// TwinCAT 3 PLC project FactoryIO
// ProgramVersion: 3.1.4024.0
// libraries:
//   Tc2_ModbusSrv, * (Beckhoff Automation GmbH)
//   Tc2_Standard, * (Beckhoff Automation GmbH)
//   Tc2_System, * (Beckhoff Automation GmbH)
//   Tc3_Module, * (Beckhoff Automation GmbH)
// project tree:
//   GVLs/ GVL.TcGVL
//   / PlcTask.TcTTO
//   POUs/FBs/Conveyor/DUTs/ E_ConveyorStates.TcDUT, ST_ConveyorConfiguration.TcDUT, ST_ConveyorControls.TcDUT, ST_ConveyorStatus.TcDUT
//   POUs/FBs/Conveyor/ FB_Conveyor.TcPOU
//   POUs/FBs/IndexedPosition/DUTs/ E_IndexedPositionSimplifiedRequest.TcDUT, E_IndexedPositionStates.TcDUT, E_IndexedPositionTransitionRequest.TcDUT, ST_DirectionalControls.TcDUT, ST_IndexedPositionControls.TcDUT, ST_IndexedPositionLinks.TcDUT
//   POUs/FBs/IndexedPosition/ FB_IndexedPosition.TcPOU
//   POUs/FBs/LTU/DUTs/ E_LTUHardwareState.TcDUT, ST_LTUConfiguration.TcDUT, ST_LTUStatus.TcDUT
//   POUs/FBs/LTU/ FB_LTU.TcPOU
//   POUs/FBs/PalletStop/DUTs/ E_PalletStopHardwareStates.TcDUT, ST_PalletStopConfiguration.TcDUT, ST_PalletStopStatus.TcDUT
//   POUs/FBs/PalletStop/ FB_PalletStop.TcPOU
//   POUs/FBs/PartPresence/DUTs/ E_ActivationType.TcDUT, ST_PartPresenceConfiguration.TcDUT, ST_PartPresenceStatus.TcDUT
//   POUs/FBs/PartPresence/ FB_PartPresence.TcPOU
//   POUs/ MAIN.TcPOU
// real-time tasks:
//   TASK PlcTask: cycle T#10ms, priority 20, ADS port 350

CONFIGURATION FactoryIO
    RESOURCE PLC ON TwinCAT3
        TASK PlcTask(INTERVAL := T#10ms, PRIORITY := 20);
        PROGRAM MAIN WITH PlcTask : MAIN;
    END_RESOURCE
END_CONFIGURATION

// ---- POUs/FBs/Conveyor/DUTs/E_ConveyorStates.TcDUT
{attribute 'qualified_only'}
{attribute 'strict'}
TYPE E_ConveyorStates :
(
	Stopped,
	RunRequest,
	Running,
	StopRequest,
	Fault
);
END_TYPE

// ---- POUs/FBs/Conveyor/DUTs/ST_ConveyorConfiguration.TcDUT
TYPE ST_ConveyorConfiguration :
	STRUCT
		Name 				: STRING := 'Conveyor'; 	// Name of the conveyor
		HardwareOutput 		: DINT;						// What position in the TCP/IP array this Bit is connected to for the simulationm
		OutputArrayPosition	: DINT;						// Equal to HardwareOutput - 32768
	END_STRUCT
END_TYPE

// ---- POUs/FBs/Conveyor/DUTs/ST_ConveyorControls.TcDUT
TYPE ST_ConveyorControls :
	STRUCT
		RequestRun 		: BOOL := FALSE; // Requests the conveyance to run
		RequestStop		: BOOL := FALSE; // Requests the conveyance to stop
		OperationMode	: BOOL := FALSE; // TRUE = Automatic, FALSE = Manual 
	END_STRUCT
END_TYPE

// ---- POUs/FBs/Conveyor/DUTs/ST_ConveyorStatus.TcDUT
TYPE ST_ConveyorStatus :
	STRUCT
		isRunning	: BOOL;  // This varriable will be True when the conveyor is running and False when it is not running
	END_STRUCT
END_TYPE

// ---- POUs/FBs/IndexedPosition/DUTs/E_IndexedPositionSimplifiedRequest.TcDUT
{attribute 'qualified_only'}
{attribute 'strict'}
TYPE E_IndexedPositionSimplifiedRequest :
(
	NoRequest,
	Busy,
	Send,
	Recieve
);
END_TYPE

// ---- POUs/FBs/IndexedPosition/DUTs/E_IndexedPositionStates.TcDUT
{attribute 'qualified_only'}
{attribute 'strict'}
TYPE E_IndexedPositionStates :
(
	Starved,
	Idle,
	Blocked,
	ReceivingFromLeft,
	ReceivingFromRight,
	ReceivingFromFront,
	ReceivingFromRear,
	SendingToLeft,
	SendingToRight,
	SendingToFront,
	SendingToRear,
	Bypass,
	Fault
);
END_TYPE

// ---- POUs/FBs/IndexedPosition/DUTs/E_IndexedPositionTransitionRequest.TcDUT
{attribute 'qualified_only'}
{attribute 'strict'}
TYPE E_IndexedPositionTransitionRequest :
(
	NoRequest,
	ReceiveFromLeft,
	ReceiveFromRight,
	ReceiveFromFront,
	ReceiveFromRear,
	SendToLeft,
	SendToRight,
	SendToFront,
	SendToRear
);
END_TYPE

// ---- POUs/FBs/IndexedPosition/DUTs/ST_DirectionalControls.TcDUT
TYPE ST_DirectionalControls :
	STRUCT
		Request 			: E_IndexedPositionSimplifiedRequest;
		PartPresent 		: BOOL;
		State				: E_IndexedPositionStates := E_IndexedPositionStates.Starved;
		OperationMode		: BOOL;
		isDefined 			: BOOL;
	END_STRUCT
END_TYPE

// ---- POUs/FBs/IndexedPosition/DUTs/ST_IndexedPositionControls.TcDUT
TYPE ST_IndexedPositionControls :
	STRUCT
		// Operating modes
		OperationMode		: BOOL := FALSE; // TRUE = Automatic, FALSE = Manual
		isDefined 			: BOOL := FALSE; // Change to true if this position exists
		State				: E_IndexedPositionStates := E_IndexedPositionStates.Starved;
		Request				: E_IndexedPositionTransitionRequest := E_IndexedPositionTransitionRequest.NoRequest;
		
		// Sensing
		ArrivalDetection	: BOOL;
		AreaMonitoring		: BOOL;

		// Internal Directional Controls for Linking
		Front				: ST_DirectionalControls;
		Rear				: ST_DirectionalControls;
		Left				: ST_DirectionalControls;
		Right				: ST_DirectionalControls;
		
	END_STRUCT
END_TYPE

// ---- POUs/FBs/IndexedPosition/DUTs/ST_IndexedPositionLinks.TcDUT
TYPE ST_IndexedPositionLinks :
	STRUCT
		Front				: REFERENCE TO ST_DirectionalControls;
		Rear				: REFERENCE TO ST_DirectionalControls;
		Left				: REFERENCE TO ST_DirectionalControls;
		Right				: REFERENCE TO ST_DirectionalControls;
	END_STRUCT
END_TYPE

// ---- POUs/FBs/LTU/DUTs/E_LTUHardwareState.TcDUT
{attribute 'qualified_only'}
{attribute 'strict'}
TYPE E_LTUHardwareState :
(
	NoCommand,
	RunForward,
	RunReverse,
	RunLeft,
	RunRight
);
END_TYPE

// ---- POUs/FBs/LTU/DUTs/ST_LTUConfiguration.TcDUT
TYPE ST_LTUConfiguration :
	STRUCT
		Name 						: STRING := 'LTU'; 			// Name of the LTU
		
		ForwardHardwareOutput 		: DINT;						// What position in the TCP/IP array this Bit is connected to for the simulationm
		ReverseHardwareOutput 		: DINT;						// What position in the TCP/IP array this Bit is connected to for the simulationm
		LeftHardwareOutput 			: DINT;						// What position in the TCP/IP array this Bit is connected to for the simulationm
		RightHardwareOutput 		: DINT;						// What position in the TCP/IP array this Bit is connected to for the simulationm
		
		ForwardOutputArrayPosition	: DINT;						// Equal to associated HardwareOutput - 32768
		ReverseOutputArrayPosition	: DINT;						// Equal to associated HardwareOutput - 32768
		LeftOutputArrayPosition		: DINT;						// Equal to associated HardwareOutput - 32768
		RightOutputArrayPosition	: DINT;						// Equal to associated HardwareOutput - 32768
		
		BypassLTU					: BOOL := FALSE; 			// This will have the LTU spin forward continuousle
	END_STRUCT
END_TYPE

// ---- POUs/FBs/LTU/DUTs/ST_LTUStatus.TcDUT
TYPE ST_LTUStatus :
STRUCT
END_STRUCT
END_TYPE

// ---- POUs/FBs/PalletStop/DUTs/E_PalletStopHardwareStates.TcDUT
{attribute 'qualified_only'}
{attribute 'strict'}
TYPE E_PalletStopHardwareStates :
(
	Raised,
	Lowered,
	Raising,
	Lowering,
	Fault
);
END_TYPE

// ---- POUs/FBs/PalletStop/DUTs/ST_PalletStopConfiguration.TcDUT
TYPE ST_PalletStopConfiguration :
	STRUCT
		Name 							: STRING := 'PalletStop'; 	// Name of the PalletStop
		DownStreamHardwareOutput 		: DINT;						// What position in the TCP/IP array this Bit is connected to for the simulationm
		DownStreamOutputArrayPosition	: DINT;						// Equal to associated HardwareOutput - 32768
	END_STRUCT
END_TYPE

// ---- POUs/FBs/PalletStop/DUTs/ST_PalletStopStatus.TcDUT
TYPE ST_PalletStopStatus :
	STRUCT
	END_STRUCT
END_TYPE

// ---- POUs/FBs/PartPresence/DUTs/E_ActivationType.TcDUT
{attribute 'qualified_only'}
{attribute 'strict'}
TYPE E_ActivationType :
(
	NormallyOpen,
	NormallyClosed
);
END_TYPE

// ---- POUs/FBs/PartPresence/DUTs/ST_PartPresenceConfiguration.TcDUT
TYPE ST_PartPresenceConfiguration :
	STRUCT
		Name 			: STRING := 'Part Presence';
		ActivationType 	: E_ActivationType := E_ActivationType.NormallyOpen;
		DebounceOnTime	: TIME := T#0S;
		DebounceOffTime	: TIME := T#0S;
		
		HardwareInput 		: BOOL;			// Mapped directly from the array
	END_STRUCT
END_TYPE

// ---- POUs/FBs/PartPresence/DUTs/ST_PartPresenceStatus.TcDUT
TYPE ST_PartPresenceStatus :
	STRUCT
		isOn : BOOL;
	END_STRUCT
END_TYPE

// ---- GVLs/GVL.TcGVL
{attribute 'qualified_only'}
VAR_GLOBAL
	mb_Input_Coils : ARRAY [0..255] OF BOOL;
	mb_Output_Coils : ARRAY [0..255] OF BOOL;
	
	// initializeControls : ST_IndexedPositionControls;
END_VAR

// ---- POUs/MAIN.TcPOU
PROGRAM MAIN
VAR
	// Actuators
	Conveyors		: ARRAY [0..16] OF FB_Conveyor;
	LTUs			: ARRAY [1..6] OF FB_LTU;
	PalletStops		: ARRAY [0..32] OF FB_PalletStop;
	
	// Sensors
	PalletStop_PartPresence_DetectArrival 	: ARRAY [0..32] OF FB_PartPresence;
	PalletStop_PartPresence_AreaMonitor		: ARRAY [0..32] OF FB_PartPresence;
	LTU_PartPresence_DetectArrival 			: ARRAY [1..6] OF FB_PartPresence;
	LTU_PartPresence_AreaMonitor			: ARRAY [1..6] OF FB_PartPresence;
	
	FirstScan		: BOOL := TRUE;
	i				: DINT;
	ToggleOn		: BOOL := FALSE;
	ToggleOff		: BOOL := FALSE;
	arrayOffset		: DINT := 32768;
	
	A : BOOL := FALSE;
END_VAR

// Fill in Reset Methods
// Set up main method for Material Flow
// Set up Error Handling
// Setup Manual Controls
// Create TwinCAT HMI for Manual Controls
// Download free ignition and create scada page
// Add Logic for sensor decisions
// Add an Actuator to do something?
// Save in GIT repo
// Maybe Add Safety and Stack Lights, Safety as real virtual safety
// Difference between HMI anbd SCADA
// Maybe Add Some Ladder?
// Scada part request

M_PartPresenceSensors();
M_Conveyors();
M_PalletStops();
M_LTUs();
M_ConveyanceLogic();

// Conveyors
FOR i := 0 TO 16 BY 1 DO
	IF ToggleOn THEN
		Conveyors[i].P_Controls.RequestRun := TRUE;
	ELSIF ToggleOff THEN
		Conveyors[i].P_Controls.RequestStop := TRUE;
	END_IF
END_FOR
ToggleOn := FALSE;
ToggleOff := FALSE;

FirstScan := FALSE;

METHOD PUBLIC M_ConveyanceLogic : BOOL
VAR_INPUT
END_VAR
///////////////////////////////////////////////////////////////////////////////////////////////////////////////////////////////////
/////////////////////////////////////////////////////// Pallet Stop Linking ///////////////////////////////////////////////////////
///////////////////////////////////////////////////////////////////////////////////////////////////////////////////////////////////

// Pallet Stop 00
PalletStops[0].P_Links.Rear 	REF= PalletStops[31].P_Controls.Front;
PalletStops[0].P_Links.Front	REF= PalletStops[1].P_Controls.Rear;

// Pallet Stop 01
PalletStops[1].P_Links.Rear		REF= PalletStops[0].P_Controls.Front;
PalletStops[1].P_Links.Front 	REF= LTUs[1].P_Controls.Rear;

// Pallet Stop 02
// Skipped

// Pallet Stop 03
PalletStops[3].P_Links.Rear		REF= LTUs[1].P_Controls.Left;
PalletStops[3].P_Links.Front 	REF= PalletStops[4].P_Controls.Rear;

// Pallet Stop 04
PalletStops[4].P_Links.Rear		REF= PalletStops[3].P_Controls.Front;
PalletStops[4].P_Links.Front 	REF= PalletStops[5].P_Controls.Rear;

// Pallet Stop 05
PalletStops[5].P_Links.Rear		REF= PalletStops[4].P_Controls.Front;
PalletStops[5].P_Links.Front 	REF= PalletStops[7].P_Controls.Rear;

// Pallet Stop 06
PalletStops[6].P_Links.Rear		REF= LTUs[1].P_Controls.Front;
PalletStops[6].P_Links.Front 	REF= LTUs[2].P_Controls.Right;

// Pallet Stop 07
PalletStops[7].P_Links.Rear		REF= PalletStops[5].P_Controls.Front;
PalletStops[7].P_Links.Front 	REF= LTUs[2].P_Controls.Rear;

// Pallet Stop 08
// Skipped

// Pallet Stop 09
// Skipped

// Pallet Stop 10
PalletStops[10].P_Links.Rear	REF= LTUs[2].P_Controls.Left;
PalletStops[10].P_Links.Front 	REF= LTUs[3].P_Controls.Rear;;

// Pallet Stop 11
// Skipped

// Pallet Stop 12
PalletStops[12].P_Links.Rear	REF= LTUs[3].P_Controls.Left;
PalletStops[12].P_Links.Front 	REF= LTUs[4].P_Controls.Rear;;

// Pallet Stop 13
// Skipped

// Pallet Stop 14
PalletStops[14].P_Links.Rear	REF= LTUs[4].P_Controls.Right;
PalletStops[14].P_Links.Front 	REF= PalletStops[15].P_Controls.Rear;

// Pallet Stop 15
PalletStops[15].P_Links.Rear	REF= PalletStops[14].P_Controls.Front;
PalletStops[15].P_Links.Front 	REF= PalletStops[16].P_Controls.Rear;

// Pallet Stop 16
PalletStops[16].P_Links.Rear	REF= PalletStops[15].P_Controls.Front;
PalletStops[16].P_Links.Front 	REF= PalletStops[17].P_Controls.Rear;

// Pallet Stop 17
PalletStops[17].P_Links.Rear	REF= PalletStops[16].P_Controls.Front;
PalletStops[17].P_Links.Front 	REF= PalletStops[32].P_Controls.Rear; // 18b

// Pallet Stop 18
PalletStops[18].P_Links.Rear	REF= LTUs[3].P_Controls.Front;
PalletStops[18].P_Links.Front 	REF= LTUs[5].P_Controls.Rear;

// Pallet Stop 19
PalletStops[19].P_Links.Rear	REF= PalletStops[32].P_Controls.Front; // 18b
PalletStops[19].P_Links.Front 	REF= LTUs[6].P_Controls.Left;

// Pallet Stop 20
// Skipped

// Pallet Stop 21
PalletStops[21].P_Links.Rear	REF= LTUs[6].P_Controls.Right;
PalletStops[21].P_Links.Front 	REF= PalletStops[22].P_Controls.Rear;

IF PalletStops[21].P_Controls.ArrivalDetection THEN
	PalletStops[21].P_Controls.Request := E_IndexedPositionTransitionRequest.SendToFront;
	//PalletStops[21].P_Links.Front.Request := E_IndexedPositionTransitionRequest.ReceiveForward;
END_IF

// Pallet Stop 22
PalletStops[22].P_Links.Rear	REF= PalletStops[21].P_Controls.Front;
PalletStops[22].P_Links.Front 	REF= PalletStops[23].P_Controls.Rear;

IF PalletStops[22].P_Controls.ArrivalDetection THEN
	PalletStops[22].P_Controls.Request := E_IndexedPositionTransitionRequest.SendToFront;
	//PalletStops[22].P_Links.Front.Request := E_IndexedPositionTransitionRequest.ReceiveForward;
END_IF

// Pallet Stop 23
PalletStops[23].P_Links.Rear	REF= PalletStops[22].P_Controls.Front;
PalletStops[23].P_Links.Front 	REF= PalletStops[24].P_Controls.Rear;

IF PalletStops[23].P_Controls.ArrivalDetection THEN
	PalletStops[23].P_Controls.Request := E_IndexedPositionTransitionRequest.SendToFront;
	//PalletStops[23].P_Links.Front.Request := E_IndexedPositionTransitionRequest.ReceiveForward;
END_IF

// Pallet Stop 24
PalletStops[24].P_Links.Rear	REF= PalletStops[23].P_Controls.Front;
PalletStops[24].P_Links.Front 	REF= PalletStops[25].P_Controls.Rear;

IF PalletStops[24].P_Controls.ArrivalDetection THEN
	PalletStops[24].P_Controls.Request := E_IndexedPositionTransitionRequest.SendToFront;
	//PalletStops[24].P_Links.Front.Request := E_IndexedPositionTransitionRequest.ReceiveForward;
END_IF

// Pallet Stop 25
PalletStops[25].P_Links.Rear	REF= PalletStops[24].P_Controls.Front;
PalletStops[25].P_Links.Front 	REF= PalletStops[26].P_Controls.Rear;

IF PalletStops[25].P_Controls.ArrivalDetection THEN
	PalletStops[25].P_Controls.Request := E_IndexedPositionTransitionRequest.SendToFront;
	//PalletStops[25].P_Links.Front.Request := E_IndexedPositionTransitionRequest.ReceiveForward;
END_IF

// Pallet Stop 26
PalletStops[26].P_Links.Rear	REF= PalletStops[25].P_Controls.Front;
PalletStops[26].P_Links.Front 	REF= PalletStops[27].P_Controls.Rear;

IF PalletStops[26].P_Controls.ArrivalDetection THEN
	PalletStops[26].P_Controls.Request := E_IndexedPositionTransitionRequest.SendToFront;
	//PalletStops[26].P_Links.Front.Request := E_IndexedPositionTransitionRequest.ReceiveForward;
END_IF

// Pallet Stop 27
PalletStops[27].P_Links.Rear	REF= PalletStops[26].P_Controls.Front;
PalletStops[27].P_Links.Front 	REF= PalletStops[28].P_Controls.Rear;

IF PalletStops[27].P_Controls.ArrivalDetection THEN
	PalletStops[27].P_Controls.Request := E_IndexedPositionTransitionRequest.SendToFront;
	//PalletStops[27].P_Links.Front.Request := E_IndexedPositionTransitionRequest.ReceiveForward;
END_IF

// Pallet Stop 28
PalletStops[28].P_Links.Rear	REF= PalletStops[27].P_Controls.Front;
PalletStops[28].P_Links.Front 	REF= PalletStops[29].P_Controls.Rear;

IF PalletStops[28].P_Controls.ArrivalDetection THEN
	PalletStops[28].P_Controls.Request := E_IndexedPositionTransitionRequest.SendToFront;
	//PalletStops[28].P_Links.Front.Request := E_IndexedPositionTransitionRequest.ReceiveForward;
END_IF

// Pallet Stop 29
PalletStops[29].P_Links.Rear	REF= PalletStops[28].P_Controls.Front;
PalletStops[29].P_Links.Front 	REF= PalletStops[30].P_Controls.Rear;

IF PalletStops[29].P_Controls.ArrivalDetection THEN
	PalletStops[29].P_Controls.Request := E_IndexedPositionTransitionRequest.SendToFront;
	//PalletStops[29].P_Links.Front.Request := E_IndexedPositionTransitionRequest.ReceiveForward;
END_IF

// Pallet Stop 30
PalletStops[30].P_Links.Rear	REF= PalletStops[29].P_Controls.Front;
PalletStops[30].P_Links.Front 	REF= PalletStops[31].P_Controls.Rear;

IF PalletStops[30].P_Controls.ArrivalDetection THEN
	PalletStops[30].P_Controls.Request := E_IndexedPositionTransitionRequest.SendToFront;
	//PalletStops[30].P_Links.Front.Request := E_IndexedPositionTransitionRequest.ReceiveForward;
END_IF

// Pallet Stop 31
PalletStops[31].P_Links.Rear	REF= PalletStops[30].P_Controls.Front;
PalletStops[31].P_Links.Front 	REF= PalletStops[0].P_Controls.Rear;

IF PalletStops[31].P_Controls.ArrivalDetection THEN
	PalletStops[31].P_Controls.Request := E_IndexedPositionTransitionRequest.SendToFront;
	//PalletStops[31].P_Links.Front.Request := E_IndexedPositionTransitionRequest.ReceiveForward;
END_IF

// Pallet Stop 18b
PalletStops[32].P_Links.Rear	REF= PalletStops[17].P_Controls.Front;
PalletStops[32].P_Links.Front 	REF= PalletStops[19].P_Controls.Rear;
END_METHOD

METHOD PUBLIC M_Conveyors : BOOL
VAR_INPUT
END_VAR
IF FirstScan THEN
	// Initialize
	FOR i := 0 TO 16 BY 1 DO
		Conveyors[i].P_Configuration.Name := CONCAT('Conveyor ', DINT_TO_STRING(i));
		Conveyors[i].P_Configuration.HardwareOutput := 32771 + i;
	END_FOR
ELSE
	FOR i := 0 TO 16 BY 1 DO
		Conveyors[i](HardwareInputArray := GVL.mb_Input_Coils);
	END_FOR
END_IF
END_METHOD

METHOD PUBLIC M_LTUs : BOOL
VAR_INPUT
END_VAR
IF FirstScan THEN
	// Initialize
	FOR i := 1 TO 6 BY 1 DO
		LTUs[i].P_Configuration.Name := CONCAT('LTU ', DINT_TO_STRING(i));
		LTUs[i].P_Configuration.ForwardHardwareOutput 	:= 32790 + 1 + ((i-1)*4);
		LTUs[i].P_Configuration.ReverseHardwareOutput 	:= 32790 + 2 + ((i-1)*4);
		LTUs[i].P_Configuration.LeftHardwareOutput 		:= 32790 + 3 + ((i-1)*4);
		LTUs[i].P_Configuration.RightHardwareOutput 	:= 32790 + 4 + ((i-1)*4);
	END_FOR
ELSE
	// Update Area Monitoring and Arrival Detection
	FOR i := 1 TO 6 BY 1 DO
		LTUs[i].P_Controls.AreaMonitoring 		:= LTU_PartPresence_AreaMonitor[i].P_Status.isOn;
		LTUs[i].P_Controls.ArrivalDetection 	:= LTU_PartPresence_DetectArrival[i].P_Status.isOn;
		LTUs[i](HardwareInputArray := GVL.mb_Input_Coils);
	END_FOR
END_IF
END_METHOD

METHOD M_PalletStops : BOOL
VAR_INPUT
END_VAR
IF FirstScan THEN
	// Initialize
	FOR i := 0 TO 32 BY 1 DO
		PalletStops[i].P_Configuration.Name := CONCAT('Pallet Stop ', DINT_TO_STRING(i));
		PalletStops[i].P_Configuration.DownStreamHardwareOutput := 32818 + i;
	END_FOR
ELSE
	// Update Area Monitoring and Arrival Detection
	FOR i := 0 TO 32 BY 1 DO
		PalletStops[i].P_Controls.AreaMonitoring 	:= PalletStop_PartPresence_AreaMonitor[i].P_Status.isOn;
		PalletStops[i].P_Controls.ArrivalDetection 	:= PalletStop_PartPresence_DetectArrival[i].P_Status.isOn;
		PalletStops[i](HardwareInputArray := GVL.mb_Input_Coils);
	END_FOR
END_IF
END_METHOD

METHOD PUBLIC M_PartPresenceSensors : BOOL
PalletStop_PartPresence_DetectArrival[0].P_Configuration.HardwareInput := GVL.mb_Output_Coils[32771 - arrayOffset];
PalletStop_PartPresence_DetectArrival[1].P_Configuration.HardwareInput := GVL.mb_Output_Coils[32772 - arrayOffset];
PalletStop_PartPresence_DetectArrival[2].P_Configuration.HardwareInput := GVL.mb_Output_Coils[32773 - arrayOffset];
PalletStop_PartPresence_DetectArrival[3].P_Configuration.HardwareInput := GVL.mb_Output_Coils[32774 - arrayOffset];
PalletStop_PartPresence_DetectArrival[4].P_Configuration.HardwareInput := GVL.mb_Output_Coils[32775 - arrayOffset];
PalletStop_PartPresence_DetectArrival[5].P_Configuration.HardwareInput := GVL.mb_Output_Coils[32776 - arrayOffset];
PalletStop_PartPresence_DetectArrival[6].P_Configuration.HardwareInput := GVL.mb_Output_Coils[32777 - arrayOffset];
PalletStop_PartPresence_DetectArrival[7].P_Configuration.HardwareInput := GVL.mb_Output_Coils[32778 - arrayOffset];
PalletStop_PartPresence_DetectArrival[8].P_Configuration.HardwareInput := GVL.mb_Output_Coils[32779 - arrayOffset];
PalletStop_PartPresence_DetectArrival[9].P_Configuration.HardwareInput := GVL.mb_Output_Coils[32780 - arrayOffset];
PalletStop_PartPresence_DetectArrival[10].P_Configuration.HardwareInput := GVL.mb_Output_Coils[32781 - arrayOffset];
PalletStop_PartPresence_DetectArrival[11].P_Configuration.HardwareInput := GVL.mb_Output_Coils[32782 - arrayOffset];
PalletStop_PartPresence_DetectArrival[12].P_Configuration.HardwareInput := GVL.mb_Output_Coils[32783 - arrayOffset];
PalletStop_PartPresence_DetectArrival[13].P_Configuration.HardwareInput := GVL.mb_Output_Coils[32784 - arrayOffset];
PalletStop_PartPresence_DetectArrival[14].P_Configuration.HardwareInput := GVL.mb_Output_Coils[32785 - arrayOffset];
PalletStop_PartPresence_DetectArrival[15].P_Configuration.HardwareInput := GVL.mb_Output_Coils[32786 - arrayOffset];
PalletStop_PartPresence_DetectArrival[16].P_Configuration.HardwareInput := GVL.mb_Output_Coils[32787 - arrayOffset];
PalletStop_PartPresence_DetectArrival[17].P_Configuration.HardwareInput := GVL.mb_Output_Coils[32788 - arrayOffset];
PalletStop_PartPresence_DetectArrival[18].P_Configuration.HardwareInput := GVL.mb_Output_Coils[32789 - arrayOffset];
PalletStop_PartPresence_DetectArrival[19].P_Configuration.HardwareInput := GVL.mb_Output_Coils[32790 - arrayOffset];
PalletStop_PartPresence_DetectArrival[20].P_Configuration.HardwareInput := GVL.mb_Output_Coils[32791 - arrayOffset];
PalletStop_PartPresence_DetectArrival[21].P_Configuration.HardwareInput := GVL.mb_Output_Coils[32792 - arrayOffset];
PalletStop_PartPresence_DetectArrival[22].P_Configuration.HardwareInput := GVL.mb_Output_Coils[32793 - arrayOffset];
PalletStop_PartPresence_DetectArrival[23].P_Configuration.HardwareInput := GVL.mb_Output_Coils[32794 - arrayOffset];
PalletStop_PartPresence_DetectArrival[24].P_Configuration.HardwareInput := GVL.mb_Output_Coils[32795 - arrayOffset];
PalletStop_PartPresence_DetectArrival[25].P_Configuration.HardwareInput := GVL.mb_Output_Coils[32796 - arrayOffset];
PalletStop_PartPresence_DetectArrival[26].P_Configuration.HardwareInput := GVL.mb_Output_Coils[32797 - arrayOffset];
PalletStop_PartPresence_DetectArrival[27].P_Configuration.HardwareInput := GVL.mb_Output_Coils[32798 - arrayOffset];
PalletStop_PartPresence_DetectArrival[28].P_Configuration.HardwareInput := GVL.mb_Output_Coils[32799 - arrayOffset];
PalletStop_PartPresence_DetectArrival[29].P_Configuration.HardwareInput := GVL.mb_Output_Coils[32800 - arrayOffset];
PalletStop_PartPresence_DetectArrival[30].P_Configuration.HardwareInput := GVL.mb_Output_Coils[32801 - arrayOffset];
PalletStop_PartPresence_DetectArrival[31].P_Configuration.HardwareInput := GVL.mb_Output_Coils[32802 - arrayOffset];
PalletStop_PartPresence_DetectArrival[32].P_Configuration.HardwareInput := GVL.mb_Output_Coils[32803 - arrayOffset];

PalletStop_PartPresence_AreaMonitor[0].P_Configuration.HardwareInput := GVL.mb_Output_Coils[32807 - arrayOffset];
PalletStop_PartPresence_AreaMonitor[1].P_Configuration.HardwareInput := GVL.mb_Output_Coils[32808 - arrayOffset];
PalletStop_PartPresence_AreaMonitor[2].P_Configuration.HardwareInput := GVL.mb_Output_Coils[32809 - arrayOffset];
PalletStop_PartPresence_AreaMonitor[3].P_Configuration.HardwareInput := GVL.mb_Output_Coils[32810 - arrayOffset] OR GVL.mb_Output_Coils[32811 - arrayOffset];
PalletStop_PartPresence_AreaMonitor[4].P_Configuration.HardwareInput := GVL.mb_Output_Coils[32812 - arrayOffset] OR GVL.mb_Output_Coils[32813 - arrayOffset] OR GVL.mb_Output_Coils[32814 - arrayOffset] OR GVL.mb_Output_Coils[32815 - arrayOffset] OR GVL.mb_Output_Coils[32816 - arrayOffset];
PalletStop_PartPresence_AreaMonitor[5].P_Configuration.HardwareInput := GVL.mb_Output_Coils[32817 - arrayOffset] OR GVL.mb_Output_Coils[32818 - arrayOffset] OR GVL.mb_Output_Coils[32819 - arrayOffset] OR GVL.mb_Output_Coils[32820 - arrayOffset] OR GVL.mb_Output_Coils[32821 - arrayOffset];
PalletStop_PartPresence_AreaMonitor[6].P_Configuration.HardwareInput := GVL.mb_Output_Coils[32822 - arrayOffset] OR GVL.mb_Output_Coils[32823 - arrayOffset];
PalletStop_PartPresence_AreaMonitor[7].P_Configuration.HardwareInput := GVL.mb_Output_Coils[32824 - arrayOffset] OR GVL.mb_Output_Coils[32825 - arrayOffset];
PalletStop_PartPresence_AreaMonitor[8].P_Configuration.HardwareInput := GVL.mb_Output_Coils[32826 - arrayOffset];
PalletStop_PartPresence_AreaMonitor[9].P_Configuration.HardwareInput := GVL.mb_Output_Coils[32827 - arrayOffset];
PalletStop_PartPresence_AreaMonitor[10].P_Configuration.HardwareInput := GVL.mb_Output_Coils[32828 - arrayOffset] OR GVL.mb_Output_Coils[32829 - arrayOffset];
PalletStop_PartPresence_AreaMonitor[11].P_Configuration.HardwareInput := GVL.mb_Output_Coils[32830 - arrayOffset];
PalletStop_PartPresence_AreaMonitor[12].P_Configuration.HardwareInput := GVL.mb_Output_Coils[32831 - arrayOffset] OR GVL.mb_Output_Coils[32832 - arrayOffset];
PalletStop_PartPresence_AreaMonitor[13].P_Configuration.HardwareInput := GVL.mb_Output_Coils[32833 - arrayOffset];
PalletStop_PartPresence_AreaMonitor[14].P_Configuration.HardwareInput := GVL.mb_Output_Coils[32834 - arrayOffset];
PalletStop_PartPresence_AreaMonitor[15].P_Configuration.HardwareInput := GVL.mb_Output_Coils[32835 - arrayOffset] OR GVL.mb_Output_Coils[32836 - arrayOffset] OR GVL.mb_Output_Coils[32837 - arrayOffset] OR GVL.mb_Output_Coils[32838 - arrayOffset] OR GVL.mb_Output_Coils[32839 - arrayOffset];
PalletStop_PartPresence_AreaMonitor[16].P_Configuration.HardwareInput := GVL.mb_Output_Coils[32840 - arrayOffset];
PalletStop_PartPresence_AreaMonitor[17].P_Configuration.HardwareInput := GVL.mb_Output_Coils[32841 - arrayOffset];
PalletStop_PartPresence_AreaMonitor[18].P_Configuration.HardwareInput := GVL.mb_Output_Coils[32842 - arrayOffset] OR GVL.mb_Output_Coils[32843 - arrayOffset] OR GVL.mb_Output_Coils[32844 - arrayOffset] OR GVL.mb_Output_Coils[32845 - arrayOffset] OR GVL.mb_Output_Coils[32846 - arrayOffset];
PalletStop_PartPresence_AreaMonitor[19].P_Configuration.HardwareInput := GVL.mb_Output_Coils[32847 - arrayOffset] OR GVL.mb_Output_Coils[32848 - arrayOffset] OR GVL.mb_Output_Coils[32849 - arrayOffset] OR GVL.mb_Output_Coils[32850 - arrayOffset] OR GVL.mb_Output_Coils[32851 - arrayOffset] OR GVL.mb_Output_Coils[32852 - arrayOffset];
PalletStop_PartPresence_AreaMonitor[20].P_Configuration.HardwareInput := GVL.mb_Output_Coils[32853 - arrayOffset];
PalletStop_PartPresence_AreaMonitor[21].P_Configuration.HardwareInput := GVL.mb_Output_Coils[32854 - arrayOffset];
PalletStop_PartPresence_AreaMonitor[22].P_Configuration.HardwareInput := GVL.mb_Output_Coils[32855 - arrayOffset];
PalletStop_PartPresence_AreaMonitor[23].P_Configuration.HardwareInput := GVL.mb_Output_Coils[32856 - arrayOffset];
PalletStop_PartPresence_AreaMonitor[24].P_Configuration.HardwareInput := GVL.mb_Output_Coils[32857 - arrayOffset];
PalletStop_PartPresence_AreaMonitor[25].P_Configuration.HardwareInput := GVL.mb_Output_Coils[32858 - arrayOffset];
PalletStop_PartPresence_AreaMonitor[26].P_Configuration.HardwareInput := GVL.mb_Output_Coils[32859 - arrayOffset];
PalletStop_PartPresence_AreaMonitor[27].P_Configuration.HardwareInput := GVL.mb_Output_Coils[32860 - arrayOffset];
PalletStop_PartPresence_AreaMonitor[28].P_Configuration.HardwareInput := GVL.mb_Output_Coils[32861 - arrayOffset];
PalletStop_PartPresence_AreaMonitor[29].P_Configuration.HardwareInput := GVL.mb_Output_Coils[32862 - arrayOffset];
PalletStop_PartPresence_AreaMonitor[30].P_Configuration.HardwareInput := GVL.mb_Output_Coils[32863 - arrayOffset] OR GVL.mb_Output_Coils[32864 - arrayOffset] OR GVL.mb_Output_Coils[32865 - arrayOffset] OR GVL.mb_Output_Coils[32866 - arrayOffset] OR GVL.mb_Output_Coils[32867 - arrayOffset];
PalletStop_PartPresence_AreaMonitor[31].P_Configuration.HardwareInput := GVL.mb_Output_Coils[32868 - arrayOffset] OR GVL.mb_Output_Coils[32869 - arrayOffset] OR GVL.mb_Output_Coils[32870 - arrayOffset] OR GVL.mb_Output_Coils[32871 - arrayOffset] OR GVL.mb_Output_Coils[32872 - arrayOffset];
PalletStop_PartPresence_AreaMonitor[32].P_Configuration.HardwareInput := GVL.mb_Output_Coils[32873 - arrayOffset];

LTU_PartPresence_DetectArrival[1].P_Configuration.HardwareInput := GVL.mb_Output_Coils[32877 - arrayOffset];
LTU_PartPresence_DetectArrival[2].P_Configuration.HardwareInput := GVL.mb_Output_Coils[32878 - arrayOffset];
LTU_PartPresence_DetectArrival[3].P_Configuration.HardwareInput := GVL.mb_Output_Coils[32879 - arrayOffset];
LTU_PartPresence_DetectArrival[4].P_Configuration.HardwareInput := GVL.mb_Output_Coils[32880 - arrayOffset];
LTU_PartPresence_DetectArrival[5].P_Configuration.HardwareInput := GVL.mb_Output_Coils[32881 - arrayOffset];
LTU_PartPresence_DetectArrival[6].P_Configuration.HardwareInput := GVL.mb_Output_Coils[32882 - arrayOffset];

LTU_PartPresence_AreaMonitor[1].P_Configuration.HardwareInput := GVL.mb_Output_Coils[32886 - arrayOffset];
LTU_PartPresence_AreaMonitor[2].P_Configuration.HardwareInput := GVL.mb_Output_Coils[32887 - arrayOffset];
LTU_PartPresence_AreaMonitor[3].P_Configuration.HardwareInput := GVL.mb_Output_Coils[32888 - arrayOffset];
LTU_PartPresence_AreaMonitor[4].P_Configuration.HardwareInput := GVL.mb_Output_Coils[32889 - arrayOffset];
LTU_PartPresence_AreaMonitor[5].P_Configuration.HardwareInput := GVL.mb_Output_Coils[32890 - arrayOffset];
LTU_PartPresence_AreaMonitor[6].P_Configuration.HardwareInput := GVL.mb_Output_Coils[32891 - arrayOffset];

FOR i := 0 TO 32 BY 1 DO
	PalletStop_PartPresence_DetectArrival[i]();
	PalletStop_PartPresence_DetectArrival[i].P_Configuration.DebounceOnTime := T#250MS;
	PalletStop_PartPresence_AreaMonitor[i]();
END_FOR

FOR i := 1 TO 6 BY 1 DO
	LTU_PartPresence_DetectArrival[i]();
	LTU_PartPresence_AreaMonitor[i]();
END_FOR
END_METHOD

END_PROGRAM

// ---- POUs/FBs/Conveyor/FB_Conveyor.TcPOU
FUNCTION_BLOCK PUBLIC FB_Conveyor

VAR_IN_OUT
	HardwareInputArray : ARRAY [*] OF BOOL;		// For Actuators
END_VAR

VAR
	Configuration 	: ST_ConveyorConfiguration;
	Controls		: ST_ConveyorControls;
	Status			: ST_ConveyorStatus;
	
	InitDone 		: BOOL := FALSE;
	
	State			: DINT := E_ConveyorStates.Stopped;
	Running			: BOOL := FALSE; // Controls conveyor running, Initialized false to ensure conveyors are off on startup
END_VAR

IF NOT InitDone THEN
	M_Init();
	InitDone:= TRUE;
ELSE
	M_Cyclic();
	M_StateMachine();
END_IF

METHOD PRIVATE M_Cyclic : BOOL
Configuration.OutputArrayPosition := Configuration.HardwareOutput - 32768;
HardwareInputArray[Configuration.OutputArrayPosition] := Running;
Status.isRunning := Running;
END_METHOD

METHOD PRIVATE M_Init : BOOL
VAR
END_VAR
END_METHOD

METHOD PUBLIC M_Reset : BOOL
VAR_INPUT
END_VAR
END_METHOD

METHOD PRIVATE M_StateMachine : BOOL
CASE State OF
	E_ConveyorStates.Stopped: 
		IF Controls.RequestRun THEN
			State := E_ConveyorStates.RunRequest;
			Controls.RequestRun := FALSE;
		END_IF
		
	E_ConveyorStates.RunRequest:
		Running := TRUE;
		State := E_ConveyorStates.Running;
		
	E_ConveyorStates.Running:
		IF Controls.RequestStop THEN
			State := E_ConveyorStates.StopRequest;
			Controls.RequestStop := FALSE;
		END_IF
		
	E_ConveyorStates.StopRequest:
		Running := FALSE;
		State := E_ConveyorStates.Stopped;
		
END_CASE
END_METHOD

PROPERTY P_Configuration : REFERENCE TO ST_ConveyorConfiguration
GET // PUBLIC
P_Configuration REF= Configuration;
END_GET
END_PROPERTY

PROPERTY PUBLIC P_Controls : REFERENCE TO ST_ConveyorControls
GET // PUBLIC
P_Controls REF= Controls;
END_GET
END_PROPERTY

PROPERTY P_Status : REFERENCE TO ST_ConveyorStatus
GET
P_Status REF= Status;
END_GET
END_PROPERTY

END_FUNCTION_BLOCK

// ---- POUs/FBs/LTU/FB_LTU.TcPOU
FUNCTION_BLOCK PUBLIC FB_LTU EXTENDS FB_IndexedPosition

VAR_IN_OUT
	HardwareInputArray : ARRAY [*] OF BOOL;		// For Actuators
END_VAR

VAR
	Configuration 		: ST_LTUConfiguration;
	Status				: ST_LTUStatus;
	
	InitDone 			: BOOL := FALSE;

	LTUHardwareState	: DINT := E_LTUHardwareState.NoCommand;
END_VAR

IF NOT InitDone THEN
	M_Init();
	InitDone:= TRUE;
ELSE
	SUPER^();
	M_Cyclic();
	M_StateMachine();
END_IF

METHOD PRIVATE M_Cyclic : BOOL
VAR_INPUT
END_VAR
Controls.isDefined := TRUE; // I exist

Configuration.ForwardOutputArrayPosition 	:= Configuration.ForwardHardwareOutput - 32768;
Configuration.ReverseOutputArrayPosition 	:= Configuration.ReverseHardwareOutput - 32768;
Configuration.LeftOutputArrayPosition 		:= Configuration.LeftHardwareOutput - 32768;
Configuration.RightOutputArrayPosition 		:= Configuration.RightHardwareOutput - 32768;

HardwareInputArray[Configuration.ForwardOutputArrayPosition] 	:= SEL( LTUHardwareState = E_LTUHardwareState.RunForward, FALSE, TRUE);
HardwareInputArray[Configuration.ReverseOutputArrayPosition] 	:= SEL( LTUHardwareState = E_LTUHardwareState.RunReverse, FALSE, TRUE);
HardwareInputArray[Configuration.LeftOutputArrayPosition] 		:= SEL( LTUHardwareState = E_LTUHardwareState.RunLeft, FALSE, TRUE);
HardwareInputArray[Configuration.RightOutputArrayPosition] 		:= SEL( LTUHardwareState = E_LTUHardwareState.RunRight, FALSE, TRUE);
END_METHOD

METHOD PRIVATE M_Init : BOOL
VAR_INPUT
END_VAR
END_METHOD

METHOD PUBLIC M_Reset : BOOL
VAR_INPUT
END_VAR
END_METHOD

METHOD PRIVATE M_StateMachine : BOOL
VAR_INPUT
END_VAR
(*IF Configuration.BypassLTU THEN
	State := E_LTUStates.Bypass;
ELSE
	State := E_LTUStates.Idle;
END_IF*)

CASE SUPER^.Controls.State OF
	E_IndexedPositionStates.Starved, 
	E_IndexedPositionStates.Idle, 
	E_IndexedPositionStates.Blocked, 
	E_IndexedPositionStates.Fault:
		LTUHardwareState := E_LTUHardwareState.NoCommand;
			
	E_IndexedPositionStates.ReceivingFromRight, 
	E_IndexedPositionStates.SendingToLeft:
		LTUHardwareState := E_LTUHardwareState.RunLeft;

	E_IndexedPositionStates.ReceivingFromLeft, 
	E_IndexedPositionStates.SendingToRight:
		LTUHardwareState := E_LTUHardwareState.RunRight;

	E_IndexedPositionStates.ReceivingFromRear, 
	E_IndexedPositionStates.SendingToFront:
		LTUHardwareState := E_LTUHardwareState.RunForward;
		
	E_IndexedPositionStates.ReceivingFromFront, 
	E_IndexedPositionStates.SendingToRear:
		LTUHardwareState := E_LTUHardwareState.RunReverse;
		
	E_IndexedPositionStates.Bypass:
		LTUHardwareState := E_LTUHardwareState.RunForward;
		
END_CASE
END_METHOD

PROPERTY PUBLIC P_Configuration : REFERENCE TO ST_LTUConfiguration
GET
P_Configuration REF= Configuration;
END_GET
END_PROPERTY

PROPERTY PUBLIC P_Status : REFERENCE TO ST_LTUStatus
GET
P_Status REF= Status;
END_GET
END_PROPERTY

END_FUNCTION_BLOCK

// ---- POUs/FBs/IndexedPosition/FB_IndexedPosition.TcPOU
FUNCTION_BLOCK PUBLIC FB_IndexedPosition

VAR
	// Configuration 		: ST_IndexedPositionConfiguration;
	Controls			: ST_IndexedPositionControls;
	// Status				: ST_IndexedPositionStatus;
	Links				: ST_IndexedPositionLinks;
END_VAR

_M_StateMachine();

// Broadcast Part Presence Status
Controls.Front.PartPresent := Controls.AreaMonitoring OR Controls.ArrivalDetection;
Controls.Rear.PartPresent := Controls.AreaMonitoring OR Controls.ArrivalDetection;
Controls.Left.PartPresent := Controls.AreaMonitoring OR Controls.ArrivalDetection;
Controls.Right.PartPresent := Controls.AreaMonitoring OR Controls.ArrivalDetection;

// Broadcast State
Controls.Front.State := Controls.State;
Controls.Rear.State := Controls.State;
Controls.Right.State := Controls.State;
Controls.Left.State := Controls.State;

// Propogate Directional Controls Request to recieve to main level
(*
IF Controls.Request =  E_IndexedPositionTransitionRequest.NoRequest (*AND Controls.State = E_IndexedPositionStates.Starved *)THEN
	IF Controls.Front.Request = E_IndexedPositionSimplifiedRequest.Recieve THEN
		Controls.Request :=  E_IndexedPositionTransitionRequest.ReceiveFromFront;
	ELSIF Controls.Rear.Request = E_IndexedPositionSimplifiedRequest.Recieve THEN
		Controls.Request :=  E_IndexedPositionTransitionRequest.ReceiveFromRear;
	ELSIF Controls.Right.Request = E_IndexedPositionSimplifiedRequest.Recieve THEN
		Controls.Request :=  E_IndexedPositionTransitionRequest.ReceiveFromRight;
	ELSIF Controls.Left.Request = E_IndexedPositionSimplifiedRequest.Recieve THEN
		Controls.Request :=  E_IndexedPositionTransitionRequest.ReceiveFromLeft;
	END_IF
END_IF
*)

// Links.Self.State := State;

METHOD PRIVATE _M_StateMachine : BOOL
VAR_INPUT
END_VAR
(*IF Configuration.BypassIndexedPosition THEN
	Controls.State := E_IndexedPositionStates.Bypass;
ELSE
	Controls.State := E_IndexedPositionStates.Idle;
END_IF*)

CASE Controls.State OF
	E_IndexedPositionStates.Starved:
		// Command 
		Controls.Request 	:= E_IndexedPositionTransitionRequest.NoRequest;
		// Error Handling
		
		// Branch Conditions
		IF NOT Controls.AreaMonitoring AND NOT Controls.ArrivalDetection THEN
			
		   	IF __ISVALIDREF(Links.Rear) THEN
				IF Links.Rear.Request = E_IndexedPositionSimplifiedRequest.Send THEN
					Controls.State 			:= E_IndexedPositionStates.ReceivingFromRear;
					Controls.Rear.Request 	:= E_IndexedPositionSimplifiedRequest.Recieve;
					// Controls.Request	 	:= E_IndexedPositionTransitionRequest.ReceiveFromRear;
				END_IF
				
			ELSIF __ISVALIDREF(Links.Front) THEN
				IF  Links.Front.Request = E_IndexedPositionSimplifiedRequest.Send THEN
					Controls.State 			:= E_IndexedPositionStates.ReceivingFromFront;
					Controls.Front.Request 	:= E_IndexedPositionSimplifiedRequest.Recieve;
					// Controls.Request	 	:= E_IndexedPositionTransitionRequest.ReceiveFromFront;
				END_IF
			
			ELSIF __ISVALIDREF(Links.Left) THEN
				IF  Links.Left.Request = E_IndexedPositionSimplifiedRequest.Send THEN
					Controls.State 			:= E_IndexedPositionStates.ReceivingFromLeft;
					Controls.Left.Request 	:= E_IndexedPositionSimplifiedRequest.Recieve;
					// Controls.Request	 	:= E_IndexedPositionTransitionRequest.ReceiveFromLeft;
				END_IF
			
			ELSIF __ISVALIDREF(Links.Right) THEN
				IF   Links.Right.Request = E_IndexedPositionSimplifiedRequest.Send THEN
					Controls.State 			:= E_IndexedPositionStates.ReceivingFromRight;
					Controls.Right.Request 	:= E_IndexedPositionSimplifiedRequest.Recieve;
					// Controls.Request	 	:= E_IndexedPositionTransitionRequest.ReceiveFromRight;
				END_IF
				
			END_IF
			
		ELSIF Controls.AreaMonitoring AND Controls.Request = E_IndexedPositionTransitionRequest.NoRequest THEN
			Controls.State 			:= E_IndexedPositionStates.Idle;
			// Controls.Request	 	:= E_IndexedPositionTransitionRequest.NoRequest;
		END_IF
		
	E_IndexedPositionStates.Idle:
			
		// Error Handling
		
		// Branch Conditions
		IF Controls.AreaMonitoring AND Controls.ArrivalDetection THEN
			// Link Request for Handshake
			IF Controls.Request = E_IndexedPositionTransitionRequest.SendToFront THEN
				Controls.Front.Request := E_IndexedPositionSimplifiedRequest.Send;
			ELSIF Controls.Request = E_IndexedPositionTransitionRequest.SendToLeft THEN
				Controls.Left.Request 	:= E_IndexedPositionSimplifiedRequest.Send;
			ELSIF Controls.Request = E_IndexedPositionTransitionRequest.SendToRear THEN
				Controls.Rear.Request 	:= E_IndexedPositionSimplifiedRequest.Send;
			ELSIF Controls.Request = E_IndexedPositionTransitionRequest.SendToRight THEN
				Controls.Right.Request := E_IndexedPositionSimplifiedRequest.Send;
			END_IF
		
			IF Controls.Request = E_IndexedPositionTransitionRequest.SendToFront THEN
				IF __ISVALIDREF(Links.Front) THEN
					IF NOT Links.Front.PartPresent AND
					   Links.Front.Request = E_IndexedPositionSimplifiedRequest.Recieve THEN
						  
						Controls.State 			:= E_IndexedPositionStates.SendingToFront;
						Controls.Front.Request 	:= E_IndexedPositionSimplifiedRequest.NoRequest;
						Links.Front.Request 	:= E_IndexedPositionSimplifiedRequest.NoRequest;
						
					ELSIF Links.Front.PartPresent OR 
						  Links.Front.Request <> E_IndexedPositionSimplifiedRequest.Recieve OR
						  Links.Front.State <> E_IndexedPositionStates.Starved THEN
						  
						Controls.State := E_IndexedPositionStates.Blocked;
						
					END_IF
				END_IF
			
			ELSIF Controls.Request = E_IndexedPositionTransitionRequest.SendToLeft THEN
				IF __ISVALIDREF(Links.Left) THEN
					IF NOT Links.Left.PartPresent AND 
						  Links.Left.Request = E_IndexedPositionSimplifiedRequest.Recieve THEN
						  
						Controls.State 			:= E_IndexedPositionStates.SendingToLeft;
						Controls.Left.Request 	:= E_IndexedPositionSimplifiedRequest.NoRequest;
						Links.Left.Request 		:= E_IndexedPositionSimplifiedRequest.NoRequest;
						
					ELSIF Links.Left.PartPresent OR 
						  Links.Left.Request <> E_IndexedPositionSimplifiedRequest.Recieve OR
						  Links.Left.State <> E_IndexedPositionStates.Starved THEN
						  
						Controls.State := E_IndexedPositionStates.Blocked;
						
					END_IF
				END_IF
				
			ELSIF Controls.Request = E_IndexedPositionTransitionRequest.SendToRear THEN
				IF __ISVALIDREF(Links.Rear) THEN
					IF NOT Links.Rear.PartPresent AND
					   Links.Rear.Request = E_IndexedPositionSimplifiedRequest.Recieve THEN
						  
						Controls.State 			:= E_IndexedPositionStates.SendingToRear;
						Controls.Rear.Request 	:= E_IndexedPositionSimplifiedRequest.NoRequest;
						Links.Rear.Request 		:= E_IndexedPositionSimplifiedRequest.NoRequest;
						
					ELSIF Links.Rear.PartPresent OR 
						  Links.Rear.Request <> E_IndexedPositionSimplifiedRequest.Recieve OR 
						  Links.Rear.State <> E_IndexedPositionStates.Starved THEN
						  
						Controls.State := E_IndexedPositionStates.Blocked;
						
					END_IF
				END_IF
				
			ELSIF Controls.Request = E_IndexedPositionTransitionRequest.SendToRight THEN
				IF __ISVALIDREF(Links.Right) THEN
					IF NOT Links.Right.PartPresent AND
					   Links.Right.Request = E_IndexedPositionSimplifiedRequest.Recieve THEN
						  
						Controls.State 			:= E_IndexedPositionStates.SendingToRight;
						Controls.Right.Request 	:= E_IndexedPositionSimplifiedRequest.NoRequest;
						Links.Right.Request 	:= E_IndexedPositionSimplifiedRequest.NoRequest;
						
					ELSIF Links.Right.PartPresent OR 
						  Links.Right.Request <> E_IndexedPositionSimplifiedRequest.Recieve OR
						  Links.Right.State <> E_IndexedPositionStates.Starved THEN
						  
						Controls.State := E_IndexedPositionStates.Blocked;
						
					END_IF
				END_IF
				
			END_IF
			
		ELSIF NOT Controls.AreaMonitoring AND NOT Controls.ArrivalDetection AND Controls.Request = E_IndexedPositionTransitionRequest.NoRequest THEN
			Controls.State 		:= E_IndexedPositionStates.Starved;
			Controls.Request 	:= E_IndexedPositionTransitionRequest.NoRequest;
			
		ELSIF Controls.AreaMonitoring OR Controls.ArrivalDetection  THEN
			//
		END_IF
	
	E_IndexedPositionStates.Blocked:
		// Command
		// Controls.Request 	:= E_IndexedPositionTransitionRequest.NoRequest;
		// Error Handling
		
		// Branch Conditions
		IF Controls.AreaMonitoring AND Controls.ArrivalDetection  THEN
			IF __ISVALIDREF(Links.Front) THEN
				IF Controls.Request = E_IndexedPositionTransitionRequest.SendToFront AND 
				   NOT Links.Front.PartPresent AND 
				   Links.Front.Request = E_IndexedPositionSimplifiedRequest.Recieve THEN
						
				   	Controls.State := E_IndexedPositionStates.Idle;
				END_IF
				
			ELSIF __ISVALIDREF(Links.Left) THEN
				IF Controls.Request = E_IndexedPositionTransitionRequest.SendToLeft AND 
			       NOT Links.Left.PartPresent AND 
				   Links.Left.Request = E_IndexedPositionSimplifiedRequest.Recieve THEN
				  
					Controls.State := E_IndexedPositionStates.Idle;
				END_IF
				
			ELSIF __ISVALIDREF(Links.Rear) THEN
				IF Controls.Request = E_IndexedPositionTransitionRequest.SendToRear AND 
			       NOT Links.Rear.PartPresent AND 
				   Links.Rear.Request = E_IndexedPositionSimplifiedRequest.Recieve THEN
				  
					Controls.State := E_IndexedPositionStates.Idle;
				END_IF
				
			ELSIF __ISVALIDREF(Links.Right) THEN
				IF Controls.Request = E_IndexedPositionTransitionRequest.SendToRight AND 
			       NOT Links.Right.PartPresent AND 
				   Links.Right.Request = E_IndexedPositionSimplifiedRequest.Recieve THEN
				  
					Controls.State := E_IndexedPositionStates.Idle;
				END_IF
				
			END_IF
			
		ELSIF NOT Controls.AreaMonitoring AND NOT Controls.ArrivalDetection  THEN
			// Starved or Error?
		END_IF
	
	E_IndexedPositionStates.ReceivingFromLeft,
	E_IndexedPositionStates.ReceivingFromRight,
	E_IndexedPositionStates.ReceivingFromFront,
	E_IndexedPositionStates.ReceivingFromRear:
		// Command
		
		// Error Handling
		
		// Branch Conditions
		IF Controls.ArrivalDetection THEN
			Controls.State 		:= E_IndexedPositionStates.Idle;
		END_IF
	
	E_IndexedPositionStates.SendingToLeft:
		// Command
		
		// Error Handling
		
		// Branch Conditions
		IF __ISVALIDREF(Links.Left) THEN
			IF Links.Left.State = E_IndexedPositionStates.Idle THEN
				Controls.State 		:= E_IndexedPositionStates.Starved;
			END_IF
		END_IF
	
	E_IndexedPositionStates.SendingToRight:
		// Command
		
		// Error Handling
		
		// Branch Conditions
		IF __ISVALIDREF(Links.Right) THEN
			IF Links.Right.State = E_IndexedPositionStates.Idle THEN
				Controls.State 		:= E_IndexedPositionStates.Starved;
			END_IF
		END_IF
		
	E_IndexedPositionStates.SendingToFront:
		// Command
		
		// Error Handling
		
		// Branch Conditions
		IF __ISVALIDREF(Links.Front) THEN
			IF Links.Front.State = E_IndexedPositionStates.Idle THEN
				Controls.State 		:= E_IndexedPositionStates.Starved;
			END_IF
		END_IF
		
	E_IndexedPositionStates.SendingToRear:
		// Command
		
		// Error Handling
		
		// Branch Conditions
		IF __ISVALIDREF(Links.Rear) THEN
			IF Links.REar.State = E_IndexedPositionStates.Idle THEN
				Controls.State 		:= E_IndexedPositionStates.Starved;
			END_IF
		END_IF
		
	E_IndexedPositionStates.Bypass:
		Controls.Request := E_IndexedPositionTransitionRequest.NoRequest;
		
	E_IndexedPositionStates.Fault:
		// Command
		Controls.Request := E_IndexedPositionTransitionRequest.NoRequest;
		
		// Error Handling
		
		// Branch Conditions
	
END_CASE
END_METHOD

PROPERTY PUBLIC P_Controls : REFERENCE TO ST_IndexedPositionControls
GET
P_Controls REF= Controls;
END_GET
END_PROPERTY

PROPERTY PUBLIC P_Links : REFERENCE TO ST_IndexedPositionLinks
GET
P_Links REF= Links;
END_GET
END_PROPERTY

END_FUNCTION_BLOCK

// ---- POUs/FBs/PalletStop/FB_PalletStop.TcPOU
FUNCTION_BLOCK PUBLIC FB_PalletStop EXTENDS FB_IndexedPosition

VAR_IN_OUT
	HardwareInputArray 	: ARRAY [*] OF BOOL;		// For Actuators
	//Upstream			: DWORD;
	//Downstream			: DWORD;
END_VAR

VAR
	Configuration 			: ST_PalletStopConfiguration;
	Status					: ST_PalletStopStatus;
	InitDone 				: BOOL := FALSE;
	PalletStopHardwareState	: DINT := E_PalletStopHardwareStates.Lowered;
END_VAR

IF NOT InitDone THEN
	M_Init();
	InitDone:= TRUE;
ELSE
	SUPER^();
	M_Cyclic();
	M_StateMachine();
END_IF

METHOD PRIVATE M_Cyclic : BOOL
VAR_INPUT
END_VAR
Controls.isDefined := TRUE; // I exist
Configuration.DownstreamOutputArrayPosition 	:= Configuration.DownstreamHardwareOutput - 32768;
HardwareInputArray[Configuration.DownstreamOutputArrayPosition] 	:= SEL( PalletStopHardwareState = E_PalletStopHardwareStates.Raised OR PalletStopHardwareState = E_PalletStopHardwareStates.Raising, FALSE, TRUE);
END_METHOD

METHOD PRIVATE M_Init : BOOL
VAR_INPUT
END_VAR
END_METHOD

METHOD PRIVATE M_StateMachine : BOOL
VAR_INPUT
END_VAR
(*IF Configuration.BypassLTU THEN
	State := E_LTUStates.Bypass;
ELSE
	State := E_LTUStates.Idle;
END_IF*)

CASE SUPER^.Controls.State OF 
// Would be better as a raise and lower requestr, followed by sensor confirmation that the Pallet Stop was raised or lowered, but no feedback from the simulation :(
	E_IndexedPositionStates.ReceivingFromRear, E_IndexedPositionStates.Idle:
		PalletStopHardwareState := E_PalletStopHardwareStates.Raised;
		
	E_IndexedPositionStates.SendingToFront, E_IndexedPositionStates.Starved:
		PalletStopHardwareState := E_PalletStopHardwareStates.Lowered;
		
END_CASE
END_METHOD

PROPERTY PUBLIC P_Configuration : REFERENCE TO ST_PalletStopConfiguration
GET
P_Configuration REF= Configuration;
END_GET
END_PROPERTY

PROPERTY PUBLIC P_Status : REFERENCE TO ST_PalletStopStatus
GET
P_Status REF= Status;
END_GET
END_PROPERTY

END_FUNCTION_BLOCK

// ---- POUs/FBs/PartPresence/FB_PartPresence.TcPOU
FUNCTION_BLOCK PUBLIC FB_PartPresence

VAR_IN_OUT
	HardwareOutputArray : ARRAY [*] OF BOOL; 	// For Sensors
END_VAR

VAR
	Configuration 		: ST_PartPresenceConfiguration;
	Status				: ST_PartPresenceStatus;
	
	InitDone 			: BOOL := FALSE;
	
	OnTimer				: TON;
	OffTimer			: TON;
END_VAR

IF NOT InitDone THEN
	M_Init();
	InitDone:= TRUE;
ELSE
	M_Cyclic();
END_IF

METHOD PRIVATE M_Cyclic : BOOL
VAR_INPUT
END_VAR
IF Configuration.ActivationType = E_ActivationType.NormallyOpen THEN
	OnTimer.IN := Configuration.HardwareInput;
	OnTimer.PT := Configuration.DebounceOnTime;
	
	OffTimer.IN := NOT Configuration.HardwareInput;
	OffTimer.PT := Configuration.DebounceOffTime;
	
ELSIF Configuration.ActivationType = E_ActivationType.NormallyClosed THEN
	OnTimer.IN := NOT Configuration.HardwareInput;
	OnTimer.PT := Configuration.DebounceOnTime;
	
	OffTimer.IN := Configuration.HardwareInput;
	OffTimer.PT := Configuration.DebounceOffTime;
END_IF

OnTimer();
OffTimer();

IF OnTimer.Q THEN
	Status.isOn := TRUE;
ELSIF OffTimer.Q THEN
	Status.isOn := FALSE;
END_IF
END_METHOD

METHOD PRIVATE M_Init : BOOL
VAR_INPUT
END_VAR
END_METHOD

METHOD PUBLIC M_Reset : BOOL
VAR_INPUT
END_VAR
END_METHOD

PROPERTY PUBLIC P_Configuration : REFERENCE TO ST_PartPresenceConfiguration
GET
P_Configuration REF= Configuration;
END_GET
END_PROPERTY

PROPERTY PUBLIC P_Status : REFERENCE TO ST_PartPresenceStatus
GET
P_Status REF= Status;
END_GET
END_PROPERTY

END_FUNCTION_BLOCK
